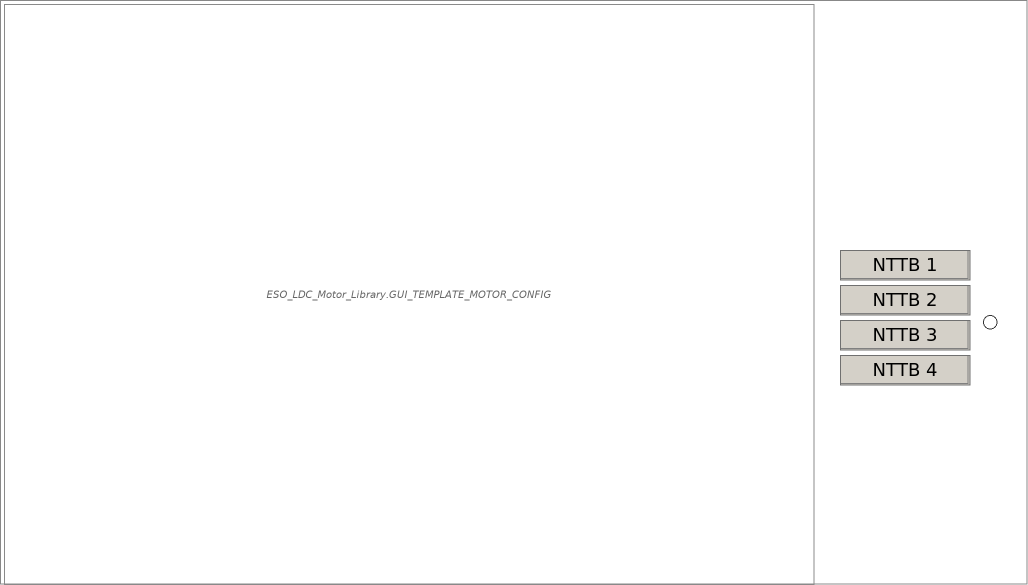
VISUALIZATION GUI_NOTT_TILT_B_CONFIG  // 1028x585
    Frame (4,4 810x581)
        shows ESO_LDC_Motor_Library.GUI_TEMPLATE_MOTOR_CONFIG(m_Instance := MAIN.nott_ics.TipTilt.ptrTiltActuatorsB[MAIN.nott_ics.TipTilt.guiTiltActuatorsBIndex]^)
    RadioButton (981,252 47x140), variable: MAIN.nott_ics.TipTilt.guiTiltActuatorsBIndex-1
        Areas[0]: Text=Radiobutton
        Areas[1]: Text=Radiobutton
    Button (840,250 130x30), "NTTB 1"
        OnMouseClick: execute { MAIN.nott_ics.TipTilt.guiTiltActuatorsBIndex := 1; }
    Button (840,285 130x30), "NTTB 2"
        OnMouseClick: execute { MAIN.nott_ics.TipTilt.guiTiltActuatorsBIndex := 2; }
    Button (840,320 130x30), "NTTB 3"
        OnMouseClick: execute { MAIN.nott_ics.TipTilt.guiTiltActuatorsBIndex := 3; }
    Button (840,355 130x30), "NTTB 4"
        OnMouseClick: execute { MAIN.nott_ics.TipTilt.guiTiltActuatorsBIndex := 4; }
END_VISUALIZATION

(* stored: Version 1.1.0.1, ProductVersion 3.1.4024.12
   Visu GUI_NOTT_TILT_B_CONFIG: Id {fea3d94e-df6a-426b-b1b0-4ee2ed845eb9} *)
